// TIA Portal V17 export
// export: Created 2023-12-22T15:08:00.1856808Z, ExportSetting WithDefaults, DisplayName Totally Integrated Automation Portal, DisplayVersion V17, DisplayName TIA Portal Openness, DisplayVersion V17, DisplayName TIA Portal Version Control Interface, DisplayVersion V17, DisplayName STEP 7 Professional, DisplayVersion V17, DisplayName STEP 7 Safety, DisplayVersion V17, DisplayName WinCC Advanced, DisplayVersion V17
FUNCTION_BLOCK "PS_Main"   // FB10, LAD
{ S7_Optimized_Access := 'FALSE' }
VERSION : 0.1
// stored: AutoNumber false, IsIECCheckEnabled false, SetENOAutomatically false, UDAEnableTagReadback false
   VAR_IN_OUT
      PS_REQ : Int;   // Требуемуе кол-во насосов
      PS_cnt : Int;
   END_VAR
   VAR DB_SPECIFIC
      Step_Up { S7_SetPoint := 'True'} : Array[1..6] of Real;   // Ускорения насоса, Гц/сек
      Step_Down { S7_SetPoint := 'True'} : Array[1..6] of Real;   // Замедление насоса, Гц/сек
   END_VAR
   VAR
      PS_One { S7_SetPoint := 'True'} : Array[0..10] of "PS_One";   // Pump System - One Pump
   END_VAR
   VAR DB_SPECIFIC
      PS_All { S7_SetPoint := 'True'} : Int := 7;   // Общее количество насосов
      PS_Group { S7_SetPoint := 'True'} : Int := 5;   // Число основных насосов
      PS_Reserv { S7_SetPoint := 'True'} : Int := 2;   // Число резервных насосов
      PS_Ready : Int;   // Число готовых насосов
      PS_CMD : Int;   // Число насосов в работе
      PS_Work : Int;   // Число штатно работающих насосов
      PS_Load : Int;   // Число нагруженных насосов
      PS_SP_Hz : Real;   // Уставка - штатная работа
      PS_Point : Real;
      PS_min_cnt : Int;   // Число замедленных насосов
   END_VAR
   VAR_TEMP   // added for the SCL form of the ladder/FBD networks
      _w1 : Bool;
   END_VAR
BEGIN

REGION Network 1: Распределение нагрузки по насосам
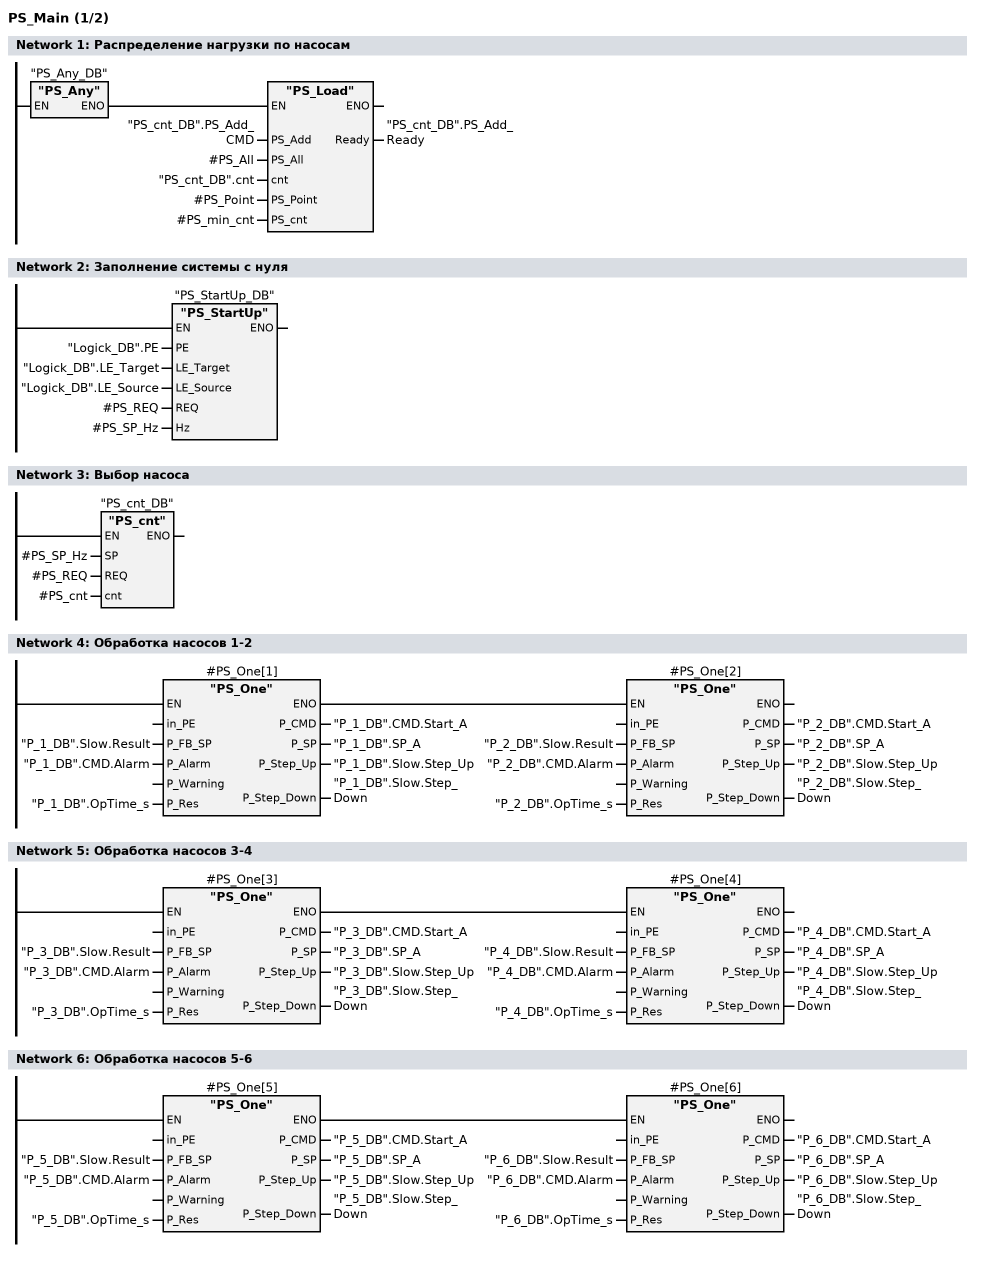
   RUNG wire#powerrail
      "PS_Any_DB"()
      "PS_Load"(PS_Add := "PS_cnt_DB".PS_Add_CMD, PS_All := #PS_All, cnt := "PS_cnt_DB".cnt, PS_Point := #PS_Point, PS_cnt := #PS_min_cnt, Ready => "PS_cnt_DB".PS_Add_Ready)
   END_RUNG
   // the same network as SCL:
   "PS_Any_DB"(ENO => #_w1);   // "PS_Any"
   IF #_w1 THEN
       "PS_Load"(PS_Add := "PS_cnt_DB".PS_Add_CMD,
                 PS_All := #PS_All,
                 cnt := "PS_cnt_DB".cnt,
                 PS_Point := #PS_Point,
                 PS_cnt := #PS_min_cnt,
                 Ready => "PS_cnt_DB".PS_Add_Ready);
   END_IF;
END_REGION

REGION Network 2: Заполнение системы с нуля
   RUNG wire#powerrail
      "PS_StartUp_DB"(PE := "Logick_DB".PE, LE_Target := "Logick_DB".LE_Target, LE_Source := "Logick_DB".LE_Source, REQ := #PS_REQ, Hz := #PS_SP_Hz)
   END_RUNG
   // the same network as SCL:
   "PS_StartUp_DB"(PE := "Logick_DB".PE,   // "PS_StartUp"
                   LE_Target := "Logick_DB".LE_Target,
                   LE_Source := "Logick_DB".LE_Source,
                   REQ := #PS_REQ,
                   Hz := #PS_SP_Hz);
END_REGION

REGION Network 3: Выбор насоса
   RUNG wire#powerrail
      "PS_cnt_DB"(SP := #PS_SP_Hz, REQ := #PS_REQ, cnt := #PS_cnt)
   END_RUNG
   // the same network as SCL:
   "PS_cnt_DB"(SP := #PS_SP_Hz, REQ := #PS_REQ, cnt := #PS_cnt);   // "PS_cnt"
END_REGION

REGION Network 4: Обработка насосов 1-2
   RUNG wire#powerrail
      #PS_One[1](in_PE :=, P_FB_SP := "P_1_DB".Slow.Result, P_Alarm := "P_1_DB".CMD.Alarm, P_Warning :=, P_Res := "P_1_DB".OpTime_s, P_CMD => "P_1_DB".CMD.Start_A, P_SP => "P_1_DB".SP_A, P_Step_Up => "P_1_DB".Slow.Step_Up, P_Step_Down => "P_1_DB".Slow.Step_Down)
      #PS_One[2](in_PE :=, P_FB_SP := "P_2_DB".Slow.Result, P_Alarm := "P_2_DB".CMD.Alarm, P_Warning :=, P_Res := "P_2_DB".OpTime_s, P_CMD => "P_2_DB".CMD.Start_A, P_SP => "P_2_DB".SP_A, P_Step_Up => "P_2_DB".Slow.Step_Up, P_Step_Down => "P_2_DB".Slow.Step_Down)
   END_RUNG
   // the same network as SCL:
   #PS_One[1](P_FB_SP := "P_1_DB".Slow.Result,   // "PS_One"
              P_Alarm := "P_1_DB".CMD.Alarm,
              P_Res := "P_1_DB".OpTime_s,
              P_CMD => "P_1_DB".CMD.Start_A,
              P_SP => "P_1_DB".SP_A,
              P_Step_Up => "P_1_DB".Slow.Step_Up,
              P_Step_Down => "P_1_DB".Slow.Step_Down,
              ENO => #_w1);
   IF #_w1 THEN
       #PS_One[2](P_FB_SP := "P_2_DB".Slow.Result,   // "PS_One"
                  P_Alarm := "P_2_DB".CMD.Alarm,
                  P_Res := "P_2_DB".OpTime_s,
                  P_CMD => "P_2_DB".CMD.Start_A,
                  P_SP => "P_2_DB".SP_A,
                  P_Step_Up => "P_2_DB".Slow.Step_Up,
                  P_Step_Down => "P_2_DB".Slow.Step_Down);
   END_IF;
END_REGION

REGION Network 5: Обработка насосов 3-4
   RUNG wire#powerrail
      #PS_One[3](in_PE :=, P_FB_SP := "P_3_DB".Slow.Result, P_Alarm := "P_3_DB".CMD.Alarm, P_Warning :=, P_Res := "P_3_DB".OpTime_s, P_CMD => "P_3_DB".CMD.Start_A, P_SP => "P_3_DB".SP_A, P_Step_Up => "P_3_DB".Slow.Step_Up, P_Step_Down => "P_3_DB".Slow.Step_Down)
      #PS_One[4](in_PE :=, P_FB_SP := "P_4_DB".Slow.Result, P_Alarm := "P_4_DB".CMD.Alarm, P_Warning :=, P_Res := "P_4_DB".OpTime_s, P_CMD => "P_4_DB".CMD.Start_A, P_SP => "P_4_DB".SP_A, P_Step_Up => "P_4_DB".Slow.Step_Up, P_Step_Down => "P_4_DB".Slow.Step_Down)
   END_RUNG
   // the same network as SCL:
   #PS_One[3](P_FB_SP := "P_3_DB".Slow.Result,   // "PS_One"
              P_Alarm := "P_3_DB".CMD.Alarm,
              P_Res := "P_3_DB".OpTime_s,
              P_CMD => "P_3_DB".CMD.Start_A,
              P_SP => "P_3_DB".SP_A,
              P_Step_Up => "P_3_DB".Slow.Step_Up,
              P_Step_Down => "P_3_DB".Slow.Step_Down,
              ENO => #_w1);
   IF #_w1 THEN
       #PS_One[4](P_FB_SP := "P_4_DB".Slow.Result,   // "PS_One"
                  P_Alarm := "P_4_DB".CMD.Alarm,
                  P_Res := "P_4_DB".OpTime_s,
                  P_CMD => "P_4_DB".CMD.Start_A,
                  P_SP => "P_4_DB".SP_A,
                  P_Step_Up => "P_4_DB".Slow.Step_Up,
                  P_Step_Down => "P_4_DB".Slow.Step_Down);
   END_IF;
END_REGION

REGION Network 6: Обработка насосов 5-6
   RUNG wire#powerrail
      #PS_One[5](in_PE :=, P_FB_SP := "P_5_DB".Slow.Result, P_Alarm := "P_5_DB".CMD.Alarm, P_Warning :=, P_Res := "P_5_DB".OpTime_s, P_CMD => "P_5_DB".CMD.Start_A, P_SP => "P_5_DB".SP_A, P_Step_Up => "P_5_DB".Slow.Step_Up, P_Step_Down => "P_5_DB".Slow.Step_Down)
      #PS_One[6](in_PE :=, P_FB_SP := "P_6_DB".Slow.Result, P_Alarm := "P_6_DB".CMD.Alarm, P_Warning :=, P_Res := "P_6_DB".OpTime_s, P_CMD => "P_6_DB".CMD.Start_A, P_SP => "P_6_DB".SP_A, P_Step_Up => "P_6_DB".Slow.Step_Up, P_Step_Down => "P_6_DB".Slow.Step_Down)
   END_RUNG
   // the same network as SCL:
   #PS_One[5](P_FB_SP := "P_5_DB".Slow.Result,   // "PS_One"
              P_Alarm := "P_5_DB".CMD.Alarm,
              P_Res := "P_5_DB".OpTime_s,
              P_CMD => "P_5_DB".CMD.Start_A,
              P_SP => "P_5_DB".SP_A,
              P_Step_Up => "P_5_DB".Slow.Step_Up,
              P_Step_Down => "P_5_DB".Slow.Step_Down,
              ENO => #_w1);
   IF #_w1 THEN
       #PS_One[6](P_FB_SP := "P_6_DB".Slow.Result,   // "PS_One"
                  P_Alarm := "P_6_DB".CMD.Alarm,
                  P_Res := "P_6_DB".OpTime_s,
                  P_CMD => "P_6_DB".CMD.Start_A,
                  P_SP => "P_6_DB".SP_A,
                  P_Step_Up => "P_6_DB".Slow.Step_Up,
                  P_Step_Down => "P_6_DB".Slow.Step_Down);
   END_IF;
END_REGION

REGION Network 7: Обработка насосов 7-8
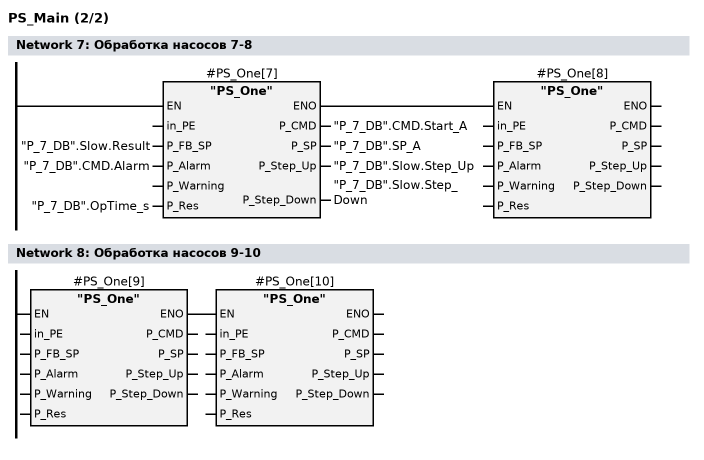
   RUNG wire#powerrail
      #PS_One[7](in_PE :=, P_FB_SP := "P_7_DB".Slow.Result, P_Alarm := "P_7_DB".CMD.Alarm, P_Warning :=, P_Res := "P_7_DB".OpTime_s, P_CMD => "P_7_DB".CMD.Start_A, P_SP => "P_7_DB".SP_A, P_Step_Up => "P_7_DB".Slow.Step_Up, P_Step_Down => "P_7_DB".Slow.Step_Down)
      #PS_One[8](in_PE :=, P_FB_SP :=, P_Alarm :=, P_Warning :=, P_Res :=, P_CMD =>, P_SP =>, P_Step_Up =>, P_Step_Down =>)
   END_RUNG
   // the same network as SCL:
   #PS_One[7](P_FB_SP := "P_7_DB".Slow.Result,   // "PS_One"
              P_Alarm := "P_7_DB".CMD.Alarm,
              P_Res := "P_7_DB".OpTime_s,
              P_CMD => "P_7_DB".CMD.Start_A,
              P_SP => "P_7_DB".SP_A,
              P_Step_Up => "P_7_DB".Slow.Step_Up,
              P_Step_Down => "P_7_DB".Slow.Step_Down,
              ENO => #_w1);
   IF #_w1 THEN
       #PS_One[8]();   // "PS_One"
   END_IF;
END_REGION

REGION Network 8: Обработка насосов 9-10
   RUNG wire#powerrail
      #PS_One[9](P_FB_SP :=, P_Alarm :=, P_Warning :=, P_Res :=, P_CMD =>, P_SP =>, P_Step_Up =>, P_Step_Down =>, in_PE :=)
      #PS_One[10](P_FB_SP :=, P_Alarm :=, P_Warning :=, P_Res :=, P_CMD =>, P_SP =>, P_Step_Up =>, P_Step_Down =>, in_PE :=)
   END_RUNG
   // the same network as SCL:
   #PS_One[9](ENO => #_w1);   // "PS_One"
   IF #_w1 THEN
       #PS_One[10]();   // "PS_One"
   END_IF;
END_REGION
END_FUNCTION_BLOCK
